(* Logix 5000 project; controller LogixAlarmExhvTest vendor 1 type 14 code 164 rev 32.11; software revision 32.03 *)

TASK MainTask (continuous, watchdog 500 ms) : MainProgram

MODULES
   Local : vendor 1 type 14 code 164 (ICP 0, rev 32.11)
END_MODULES

TYPE TestDataTypeForAlarm :
STRUCT
   M1 : DINT;
END_STRUCT
END_TYPE

VAR_GLOBAL   (* controller tags *)
   logixAlrTag1 : DINT;
   logixAlrTag2 : DINT;
END_VAR

PROGRAM MainProgram   (* main routine MainRoutine *)
VAR
   NewAlarmType : UINT;   // New Alarm Uint
   Timer : TIMER;
END_VAR

ROUTINE MainRoutine   (* ladder *)
   0: ;
END_ROUTINE
END_PROGRAM
